FUNCTION_BLOCK FB_PickAndPlace_SFC EXTENDS FB_Controller_SFC
VAR_INPUT
	Mover: BOOL;
	TPIN: TIME; (* Tiempo de cierre y apertura de la pinza de carga *)	
	h0: BOOL; 	(* Final de carrera horizontal retraida *)
	h1: BOOL; 	(* Final de carrera horizontal extendido *)
	v1: BOOL; 	(*Final de carrera vertical abajo*)
	v0: BOOL; 	(*Final de carrera vertical arriba*)
END_VAR
VAR_OUTPUT	
	HOR			: BOOL; (* Actuador de extension de brazo horizontal *)
	VER			: BOOL; (* Actuador de movimiento vertical de brazo*)
	PIN			: BOOL; (*Actuador de pinza de brazo*)
END_VAR

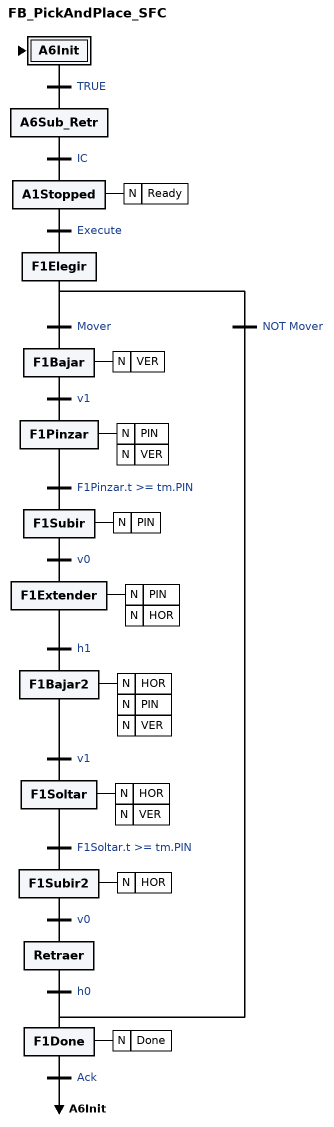
INITIAL_STEP A6Init:
END_STEP
TRANSITION FROM A6Init TO A6Sub_Retr
    := TRUE;
END_TRANSITION
STEP A6Sub_Retr:
END_STEP
TRANSITION FROM A6Sub_Retr TO A1Stopped
    := IC;
END_TRANSITION
STEP A1Stopped:
    Ready(N);
END_STEP
TRANSITION FROM A1Stopped TO F1Elegir
    := Execute;
END_TRANSITION
STEP F1Elegir:
END_STEP
TRANSITION FROM F1Elegir TO F1Bajar
    := Mover;
END_TRANSITION
STEP F1Bajar:
    VER(N);
END_STEP
TRANSITION FROM F1Bajar TO F1Pinzar
    := v1;
END_TRANSITION
STEP F1Pinzar:
    PIN(N);
    VER(N);
END_STEP
TRANSITION FROM F1Pinzar TO F1Subir
    := F1Pinzar.t >= tm.PIN;
END_TRANSITION
STEP F1Subir:
    PIN(N);
END_STEP
TRANSITION FROM F1Subir TO F1Extender
    := v0;
END_TRANSITION
STEP F1Extender:
    PIN(N);
    HOR(N);
END_STEP
TRANSITION FROM F1Extender TO F1Bajar2
    := h1;
END_TRANSITION
STEP F1Bajar2:
    HOR(N);
    PIN(N);
    VER(N);
END_STEP
TRANSITION FROM F1Bajar2 TO F1Soltar
    := v1;
END_TRANSITION
STEP F1Soltar:
    HOR(N);
    VER(N);
END_STEP
TRANSITION FROM F1Soltar TO F1Subir2
    := F1Soltar.t >= tm.PIN;
END_TRANSITION
STEP F1Subir2:
    HOR(N);
END_STEP
TRANSITION FROM F1Subir2 TO Retraer
    := v0;
END_TRANSITION
STEP Retraer:
END_STEP
TRANSITION FROM Retraer TO F1Done
    := h0;
END_TRANSITION
TRANSITION FROM F1Elegir TO F1Done
    := NOT Mover;
END_TRANSITION
STEP F1Done:
    Done(N);
END_STEP
TRANSITION FROM F1Done TO A6Init
    := Ack;
END_TRANSITION

END_FUNCTION_BLOCK

(* stored: Version 1.1.0.1, ProductVersion 3.1.4024.11
   POU FB_PickAndPlace_SFC: Id {5cf52b3a-efe0-4468-b39c-acadeafc1635}, SpecialFunc None *)
